FUNCTION_BLOCK FB_ProfilerPractice

VAR
	fbProfiler : PROFILER;
	stProfilerResult : PROFILERSTRUCT;
	nFactorial : ULINT;
	n : ULINT := 1000;
END_VAR

fbProfiler(START := TRUE, RESET := FALSE);
Factorial(n := n , nFactorialValue => nFactorial );
fbProfiler(START := FALSE);
stProfilerResult := fbProfiler.DATA;

METHOD Factorial
VAR_INPUT
	n : ULINT;
END_VAR
VAR
	nCounter : ULINT;
END_VAR
VAR_OUTPUT
	nFactorialValue : ULINT := 1;
END_VAR
FOR nCounter := 1 TO n DO
	nFactorialValue := nFactorialValue * nCounter;
END_FOR
END_METHOD

END_FUNCTION_BLOCK

(* stored: Version 1.1.0.1, ProductVersion 3.1.4024.16
   POU FB_ProfilerPractice: Id {3a919baf-a0c6-4189-ac62-1047e3e3c772}, SpecialFunc None
   Method Factorial: Id {795a7f79-0c5e-4563-8b2d-5ee31d6886a1} *)
